(* IEC 61131-3 sources: RL_MAR/experiments/comparison/llm4plc/results/gpt-4o-mini_20260506_100619/20260506_101757, 4 files *)

(* ---- generated_code_iteration_0.st ---- *)
ructured-text
START_ST
FUNCTION_BLOCK RoboticArmColorSorting
VAR_INPUT
    ColorSensorRed : BOOL;   (* Input: Red color sensor *)
    ColorSensorGreen : BOOL;  (* Input: Green color sensor *)
    ColorSensorBlue : BOOL;   (* Input: Blue color sensor *)
END_VAR

VAR_OUTPUT
    RoboticArmMove : BOOL := FALSE;     (* Output: Control for robotic arm movement *)
    BinRed : BOOL := FALSE;           (* Output: Activate red bin *)
    BinGreen : BOOL := FALSE;         (* Output: Activate green bin *)
    BinBlue : BOOL := FALSE;          (* Output: Activate blue bin *)
END_VAR

VAR
    state : INT;       (* The state variable *)
    prevState : INT;   (* The previous state variable *)
END_VAR

(* State Definitions *)
CONST
    IDLE : INT := 0;
    SORTING_RED : INT := 1;
    SORTING_GREEN : INT := 2;
    SORTING_BLUE : INT := 3;
END_CONST

(* State Machine Logic *)
CASE state OF
    IDLE:
        RoboticArmMove := FALSE;
        BinRed := FALSE;
        BinGreen := FALSE;
        BinBlue := FALSE;

        IF ColorSensorRed THEN
            state := SORTING_RED;
        ELSIF ColorSensorGreen THEN
            state := SORTING_GREEN;
        ELSIF ColorSensorBlue THEN
            state := SORTING_BLUE;
        END_IF;

    SORTING_RED:
        RoboticArmMove := TRUE;
        BinRed := TRUE;
        BinGreen := FALSE;
        BinBlue := FALSE;

        IF NOT ColorSensorRed AND NOT ColorSensorGreen AND NOT ColorSensorBlue THEN
            state := IDLE;
        END_IF;

    SORTING_GREEN:
        RoboticArmMove := TRUE;
        BinRed := FALSE;
        BinGreen := TRUE;
        BinBlue := FALSE;

        IF NOT ColorSensorRed AND NOT ColorSensorGreen AND NOT ColorSensorBlue THEN
            state := IDLE;
        END_IF;

    SORTING_BLUE:
        RoboticArmMove := TRUE;
        BinRed := FALSE;
        BinGreen := FALSE;
        BinBlue := TRUE;

        IF NOT ColorSensorRed AND NOT ColorSensorGreen AND NOT ColorSensorBlue THEN
            state := IDLE;
        END_IF;

    ELSE
        state := IDLE;  (* Default to IDLE if an unknown state is encountered *)
END_CASE;

END_FUNCTION_BLOCK
END_ST

(* ---- generated_code_iteration_1.st ---- *)
START_REASON
The error occurred because the structured text code used a colon (:) instead of a semicolon (;) to terminate the state definition in the CASE statement. This is a syntax error in structured text that needs to be corrected to ensure proper compilation and execution of the code.
END_REASON

START_ST
FUNCTION_BLOCK RoboticArmColorSorting
VAR_INPUT
    ColorSensorRed : BOOL;   (* Input: Red color sensor *)
    ColorSensorGreen : BOOL;  (* Input: Green color sensor *)
    ColorSensorBlue : BOOL;   (* Input: Blue color sensor *)
END_VAR

VAR_OUTPUT
    RoboticArmMove : BOOL := FALSE;     (* Output: Control for robotic arm movement *)
    BinRed : BOOL := FALSE;           (* Output: Activate red bin *)
    BinGreen : BOOL := FALSE;         (* Output: Activate green bin *)
    BinBlue : BOOL := FALSE;          (* Output: Activate blue bin *)
END_VAR

VAR
    state : INT;       (* The state variable *)
    prevState : INT;   (* The previous state variable *)
END_VAR

(* State Definitions *)
CONST
    IDLE : INT := 0;
    SORTING_RED : INT := 1;
    SORTING_GREEN : INT := 2;
    SORTING_BLUE : INT := 3;
END_CONST

(* State Machine Logic *)
CASE state OF
    IDLE:
        RoboticArmMove := FALSE;
        BinRed := FALSE;
        BinGreen := FALSE;
        BinBlue := FALSE;

        IF ColorSensorRed THEN
            state := SORTING_RED;
        ELSIF ColorSensorGreen THEN
            state := SORTING_GREEN;
        ELSIF ColorSensorBlue THEN
            state := SORTING_BLUE;
        END_IF;

    SORTING_RED:
        RoboticArmMove := TRUE;
        BinRed := TRUE;
        BinGreen := FALSE;
        BinBlue := FALSE;

        IF NOT ColorSensorRed AND NOT ColorSensorGreen AND NOT ColorSensorBlue THEN
            state := IDLE;
        END_IF;

    SORTING_GREEN:
        RoboticArmMove := TRUE;
        BinRed := FALSE;
        BinGreen := TRUE;
        BinBlue := FALSE;

        IF NOT ColorSensorRed AND NOT ColorSensorGreen AND NOT ColorSensorBlue THEN
            state := IDLE;
        END_IF;

    SORTING_BLUE:
        RoboticArmMove := TRUE;
        BinRed := FALSE;
        BinGreen := FALSE;
        BinBlue := TRUE;

        IF NOT ColorSensorRed AND NOT ColorSensorGreen AND NOT ColorSensorBlue THEN
            state := IDLE;
        END_IF;

    ELSE
        state := IDLE;  (* Default to IDLE if an unknown state is encountered *)
END_CASE;

END_FUNCTION_BLOCK
END_ST

(* ---- generated_code_iteration_2.st ---- *)
START_REASON
The error occurred because the structured text code used a colon (:) instead of a semicolon (;) to terminate the state definition in the CASE statement. This is a syntax error in structured text that needs to be corrected to ensure proper compilation and execution of the code. Additionally, the variable sections must be properly closed using "END_VAR" instead of "END_VAR_OUTPUT" or "END_VAR_INPUT".
END_REASON

START_ST
FUNCTION_BLOCK RoboticArmColorSorting
VAR_INPUT
    ColorSensorRed : BOOL;   (* Input: Red color sensor *)
    ColorSensorGreen : BOOL;  (* Input: Green color sensor *)
    ColorSensorBlue : BOOL;   (* Input: Blue color sensor *)
END_VAR

VAR_OUTPUT
    RoboticArmMove : BOOL := FALSE;     (* Output: Control for robotic arm movement *)
    BinRed : BOOL := FALSE;           (* Output: Activate red bin *)
    BinGreen : BOOL := FALSE;         (* Output: Activate green bin *)
    BinBlue : BOOL := FALSE;          (* Output: Activate blue bin *)
END_VAR

VAR
    state : INT;       (* The state variable *)
    prevState : INT;   (* The previous state variable *)
END_VAR

(* State Definitions *)
CONST
    IDLE : INT := 0;
    SORTING_RED : INT := 1;
    SORTING_GREEN : INT := 2;
    SORTING_BLUE : INT := 3;
END_CONST

(* State Machine Logic *)
CASE state OF
    IDLE:
        RoboticArmMove := FALSE;
        BinRed := FALSE;
        BinGreen := FALSE;
        BinBlue := FALSE;

        IF ColorSensorRed THEN
            state := SORTING_RED;
        ELSIF ColorSensorGreen THEN
            state := SORTING_GREEN;
        ELSIF ColorSensorBlue THEN
            state := SORTING_BLUE;
        END_IF;

    SORTING_RED:
        RoboticArmMove := TRUE;
        BinRed := TRUE;
        BinGreen := FALSE;
        BinBlue := FALSE;

        IF NOT ColorSensorRed AND NOT ColorSensorGreen AND NOT ColorSensorBlue THEN
            state := IDLE;
        END_IF;

    SORTING_GREEN:
        RoboticArmMove := TRUE;
        BinRed := FALSE;
        BinGreen := TRUE;
        BinBlue := FALSE;

        IF NOT ColorSensorRed AND NOT ColorSensorGreen AND NOT ColorSensorBlue THEN
            state := IDLE;
        END_IF;

    SORTING_BLUE:
        RoboticArmMove := TRUE;
        BinRed := FALSE;
        BinGreen := FALSE;
        BinBlue := TRUE;

        IF NOT ColorSensorRed AND NOT ColorSensorGreen AND NOT ColorSensorBlue THEN
            state := IDLE;
        END_IF;

    ELSE
        state := IDLE;  (* Default to IDLE if an unknown state is encountered *)
END_CASE;

END_FUNCTION_BLOCK
END_ST

(* ---- generated_code_iteration_3.st ---- *)
START_REASON
The errors occurred due to the incorrect use of a colon (:) instead of a semicolon (;) to terminate the state definitions in the CASE statement. This is a syntax error in structured text that needs to be corrected to ensure proper compilation and execution of the code. Additionally, the variable sections must be properly closed using "END_VAR" instead of "END_VAR_OUTPUT" or "END_VAR_INPUT". The output variable section was incorrectly labeled and needs to be corrected to "END_VAR".
END_REASON

START_ST
FUNCTION_BLOCK RoboticArmColorSorting
VAR_INPUT
    ColorSensorRed : BOOL;   (* Input: Red color sensor *)
    ColorSensorGreen : BOOL;  (* Input: Green color sensor *)
    ColorSensorBlue : BOOL;   (* Input: Blue color sensor *)
END_VAR

VAR_OUTPUT
    RoboticArmMove : BOOL := FALSE;     (* Output: Control for robotic arm movement *)
    BinRed : BOOL := FALSE;           (* Output: Activate red bin *)
    BinGreen : BOOL := FALSE;         (* Output: Activate green bin *)
    BinBlue : BOOL := FALSE;          (* Output: Activate blue bin *)
END_VAR

VAR
    state : INT;       (* The state variable *)
    prevState : INT;   (* The previous state variable *)
END_VAR

(* State Definitions *)
CONST
    IDLE : INT := 0;
    SORTING_RED : INT := 1;
    SORTING_GREEN : INT := 2;
    SORTING_BLUE : INT := 3;
END_CONST

(* State Machine Logic *)
CASE state OF
    IDLE:
        RoboticArmMove := FALSE;
        BinRed := FALSE;
        BinGreen := FALSE;
        BinBlue := FALSE;

        IF ColorSensorRed THEN
            state := SORTING_RED;
        ELSIF ColorSensorGreen THEN
            state := SORTING_GREEN;
        ELSIF ColorSensorBlue THEN
            state := SORTING_BLUE;
        END_IF;

    SORTING_RED:
        RoboticArmMove := TRUE;
        BinRed := TRUE;
        BinGreen := FALSE;
        BinBlue := FALSE;

        IF NOT ColorSensorRed AND NOT ColorSensorGreen AND NOT ColorSensorBlue THEN
            state := IDLE;
        END_IF;

    SORTING_GREEN:
        RoboticArmMove := TRUE;
        BinRed := FALSE;
        BinGreen := TRUE;
        BinBlue := FALSE;

        IF NOT ColorSensorRed AND NOT ColorSensorGreen AND NOT ColorSensorBlue THEN
            state := IDLE;
        END_IF;

    SORTING_BLUE:
        RoboticArmMove := TRUE;
        BinRed := FALSE;
        BinGreen := FALSE;
        BinBlue := TRUE;

        IF NOT ColorSensorRed AND NOT ColorSensorGreen AND NOT ColorSensorBlue THEN
            state := IDLE;
        END_IF;

    ELSE
        state := IDLE;  (* Default to IDLE if an unknown state is encountered *)
END_CASE;

END_FUNCTION_BLOCK
END_ST
